// TIA Portal V18 export
FUNCTION_BLOCK "NG"   // FB2901, LAD
{ S7_Optimized_Access := 'TRUE' }
// stored: AutoNumber false, MemoryReserve 100, SetENOAutomatically false
   VAR
      NG_L_1 : "NGStatus";
      NG_L_2 { S7_SetPoint := 'True'} : "NGStatus";
      NG_L_3 { S7_SetPoint := 'True'} : "NGStatus";
      NG_UL_1 { S7_SetPoint := 'True'} : "NGStatus";
      NG_UL_2 { S7_SetPoint := 'True'} : "NGStatus";
      NG_UL_3 { S7_SetPoint := 'True'} : "NGStatus";
   END_VAR
   VAR_TEMP   // added for the SCL form of the ladder/FBD networks
      _w1 : Bool;
      _w2 : Bool;
      _w3 : Bool;
      _w4 : Bool;
      _w5 : Bool;
      _w6 : Bool;
      _w7 : Bool;
      _w8 : Bool;
      _w9 : Bool;
      _w10 : Bool;
      _w11 : Bool;
      _w12 : Bool;
      _w13 : Bool;
   END_VAR
BEGIN

REGION Network 1 (SCL): Input
   // NG1
   "PalletNGData".LoadingNGPallet.NG_1_1 := "iE1-UnloadingShaftPressNG_5";
   "PalletNGData".LoadingNGPallet.NG_1_2 := "iE1-UnloadingShaftPressNG_4";
   "PalletNGData".LoadingNGPallet.NG_1_3 := "iE1-UnloadingShaftPressNG_3";
   "PalletNGData".LoadingNGPallet.NG_1_4 := "iE1-UnloadingShaftPressNG_2";
   "PalletNGData".LoadingNGPallet.NG_1_5 := "iE1-UnloadingShaftPressNG_1";

   "PalletNGData".LoadingNGPallet.NG_2_1 := "iE1-UnloadingShaftScanNG_5";
   "PalletNGData".LoadingNGPallet.NG_2_2 := "iE1-UnloadingShaftScanNG_4";
   "PalletNGData".LoadingNGPallet.NG_2_3 := "iE1-UnloadingShaftScanNG_3";
   "PalletNGData".LoadingNGPallet.NG_2_4 := "iE1-UnloadingShaftScanNG_2";
   "PalletNGData".LoadingNGPallet.NG_2_5 := "iE1-UnloadingShaftScanNG_1";

   "PalletNGData".LoadingNGPallet.NG_3_1 := "iE1-UnloadingRingScanNG_5";
   "PalletNGData".LoadingNGPallet.NG_3_2 := "iE1-UnloadingRingScanNG_4";
   "PalletNGData".LoadingNGPallet.NG_3_3 := "iE1-UnloadingRingScanNG_3";
   "PalletNGData".LoadingNGPallet.NG_3_4 := "iE1-UnloadingRingScanNG_2";
   "PalletNGData".LoadingNGPallet.NG_3_5 := "iE1-UnloadingRingScanNG_1";

   // NG2
   "PalletNGData".UnLoadingNGPallet.NG_1_1 := "iE2-UnloadingPressNG_5";
   "PalletNGData".UnLoadingNGPallet.NG_1_2 := "iE2-UnloadingPressNG_4";
   "PalletNGData".UnLoadingNGPallet.NG_1_3 := "iE2-UnloadingPressNG_3";
   "PalletNGData".UnLoadingNGPallet.NG_1_4 := "iE2-UnloadingPressNG_2";
   "PalletNGData".UnLoadingNGPallet.NG_1_5 := "iE2-UnloadingPressNG_1";

   "PalletNGData".UnLoadingNGPallet.NG_2_1 := "iE2-UnloadingMagentScanNG_5";
   "PalletNGData".UnLoadingNGPallet.NG_2_2 := "iE2-UnloadingMagentScanNG_4";
   "PalletNGData".UnLoadingNGPallet.NG_2_3 := "iE2-UnloadingMagentScanNG_3";
   "PalletNGData".UnLoadingNGPallet.NG_2_4 := "iE2-UnloadingMagentScanNG_2";
   "PalletNGData".UnLoadingNGPallet.NG_2_5 := "iE2-UnloadingMagentScanNG_1";

   "PalletNGData".UnLoadingNGPallet.NG_3_1 := "iE2-UnloadingRingScanNG_5";
   "PalletNGData".UnLoadingNGPallet.NG_3_2 := "iE2-UnloadingRingScanNG_4";
   "PalletNGData".UnLoadingNGPallet.NG_3_3 := "iE2-UnloadingRingScanNG_3";
   "PalletNGData".UnLoadingNGPallet.NG_3_4 := "iE2-UnloadingRingScanNG_2";
   "PalletNGData".UnLoadingNGPallet.NG_3_5 := "iE2-UnloadingRingScanNG_1";
END_REGION

REGION Network 2: --------------------------------------- Load -------------------------------------------------------
END_REGION

REGION Network 3: Press
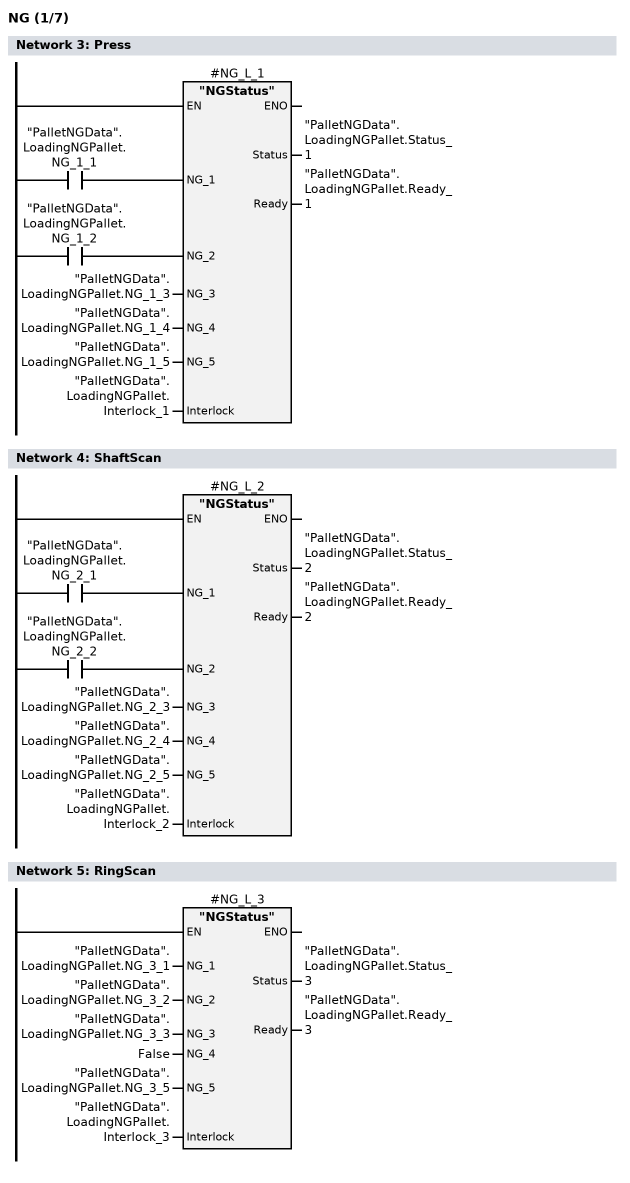
   RUNG wire#powerrail
      #NG_L_1(NG_1 := wire#w1, NG_2 := wire#w2, NG_3 := "PalletNGData".LoadingNGPallet.NG_1_3, NG_4 := "PalletNGData".LoadingNGPallet.NG_1_4, NG_5 := "PalletNGData".LoadingNGPallet.NG_1_5, Interlock := "PalletNGData".LoadingNGPallet.Interlock_1, Status => "PalletNGData".LoadingNGPallet.Status_1, Ready => "PalletNGData".LoadingNGPallet.Ready_1)
   END_RUNG
   RUNG wire#powerrail
      Contact( "PalletNGData".LoadingNGPallet.NG_1_1 )
   END_RUNG wire#w1
   RUNG wire#powerrail
      Contact( "PalletNGData".LoadingNGPallet.NG_1_2 )
   END_RUNG wire#w2
   // the same network as SCL:
   #NG_L_1(NG_1 := "PalletNGData".LoadingNGPallet.NG_1_1,   // "NGStatus"
           NG_2 := "PalletNGData".LoadingNGPallet.NG_1_2,
           NG_3 := "PalletNGData".LoadingNGPallet.NG_1_3,
           NG_4 := "PalletNGData".LoadingNGPallet.NG_1_4,
           NG_5 := "PalletNGData".LoadingNGPallet.NG_1_5,
           Interlock := "PalletNGData".LoadingNGPallet.Interlock_1,
           Status => "PalletNGData".LoadingNGPallet.Status_1,
           Ready => "PalletNGData".LoadingNGPallet.Ready_1);
END_REGION

REGION Network 4: ShaftScan
   RUNG wire#powerrail
      #NG_L_2(NG_1 := wire#w1, NG_2 := wire#w2, NG_3 := "PalletNGData".LoadingNGPallet.NG_2_3, NG_4 := "PalletNGData".LoadingNGPallet.NG_2_4, NG_5 := "PalletNGData".LoadingNGPallet.NG_2_5, Interlock := "PalletNGData".LoadingNGPallet.Interlock_2, Status => "PalletNGData".LoadingNGPallet.Status_2, Ready => "PalletNGData".LoadingNGPallet.Ready_2)
   END_RUNG
   RUNG wire#powerrail
      Contact( "PalletNGData".LoadingNGPallet.NG_2_1 )
   END_RUNG wire#w1
   RUNG wire#powerrail
      Contact( "PalletNGData".LoadingNGPallet.NG_2_2 )
   END_RUNG wire#w2
   // the same network as SCL:
   #NG_L_2(NG_1 := "PalletNGData".LoadingNGPallet.NG_2_1,   // "NGStatus"
           NG_2 := "PalletNGData".LoadingNGPallet.NG_2_2,
           NG_3 := "PalletNGData".LoadingNGPallet.NG_2_3,
           NG_4 := "PalletNGData".LoadingNGPallet.NG_2_4,
           NG_5 := "PalletNGData".LoadingNGPallet.NG_2_5,
           Interlock := "PalletNGData".LoadingNGPallet.Interlock_2,
           Status => "PalletNGData".LoadingNGPallet.Status_2,
           Ready => "PalletNGData".LoadingNGPallet.Ready_2);
END_REGION

REGION Network 5: RingScan
   RUNG wire#powerrail
      #NG_L_3(NG_1 := "PalletNGData".LoadingNGPallet.NG_3_1, NG_2 := "PalletNGData".LoadingNGPallet.NG_3_2, NG_3 := "PalletNGData".LoadingNGPallet.NG_3_3, NG_4 := False, NG_5 := "PalletNGData".LoadingNGPallet.NG_3_5, Interlock := "PalletNGData".LoadingNGPallet.Interlock_3, Status => "PalletNGData".LoadingNGPallet.Status_3, Ready => "PalletNGData".LoadingNGPallet.Ready_3)
   END_RUNG
   // the same network as SCL:
   #NG_L_3(NG_1 := "PalletNGData".LoadingNGPallet.NG_3_1,   // "NGStatus"
           NG_2 := "PalletNGData".LoadingNGPallet.NG_3_2,
           NG_3 := "PalletNGData".LoadingNGPallet.NG_3_3,
           NG_4 := False,
           NG_5 := "PalletNGData".LoadingNGPallet.NG_3_5,
           Interlock := "PalletNGData".LoadingNGPallet.Interlock_3,
           Status => "PalletNGData".LoadingNGPallet.Status_3,
           Ready => "PalletNGData".LoadingNGPallet.Ready_3);
END_REGION

REGION Network 6: InterLock
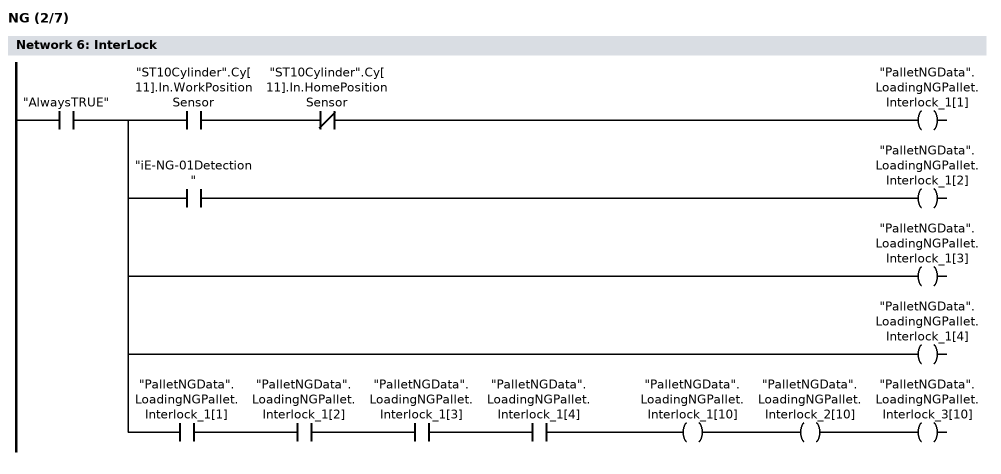
   RUNG wire#powerrail
      Contact( "AlwaysTRUE" )
      wire#w1
      Contact( "ST10Cylinder".Cy[11].In.WorkPositionSensor )
      I_Contact( "ST10Cylinder".Cy[11].In.HomePositionSensor )
      Coil( "PalletNGData".LoadingNGPallet.Interlock_1[1] )
   END_RUNG
   RUNG wire#w1
      Contact( "iE-NG-01Detection" )
      Coil( "PalletNGData".LoadingNGPallet.Interlock_1[2] )
   END_RUNG
   RUNG wire#w1
      Coil( "PalletNGData".LoadingNGPallet.Interlock_1[3] )
   END_RUNG
   RUNG wire#w1
      Coil( "PalletNGData".LoadingNGPallet.Interlock_1[4] )
   END_RUNG
   RUNG wire#w1
      Contact( "PalletNGData".LoadingNGPallet.Interlock_1[1] )
      Contact( "PalletNGData".LoadingNGPallet.Interlock_1[2] )
      Contact( "PalletNGData".LoadingNGPallet.Interlock_1[3] )
      Contact( "PalletNGData".LoadingNGPallet.Interlock_1[4] )
      Coil( "PalletNGData".LoadingNGPallet.Interlock_1[10] )
      Coil( "PalletNGData".LoadingNGPallet.Interlock_2[10] )
      Coil( "PalletNGData".LoadingNGPallet.Interlock_3[10] )
   END_RUNG
   // the same network as SCL:
   "PalletNGData".LoadingNGPallet.Interlock_1[1] := "AlwaysTRUE" AND "ST10Cylinder".Cy[11].In.WorkPositionSensor AND NOT "ST10Cylinder".Cy[11].In.HomePositionSensor;
   "PalletNGData".LoadingNGPallet.Interlock_1[2] := "AlwaysTRUE" AND "iE-NG-01Detection";
   "PalletNGData".LoadingNGPallet.Interlock_1[3] := "AlwaysTRUE";
   "PalletNGData".LoadingNGPallet.Interlock_1[4] := "AlwaysTRUE";
   #_w1 := "AlwaysTRUE" AND "PalletNGData".LoadingNGPallet.Interlock_1[1] AND "PalletNGData".LoadingNGPallet.Interlock_1[2] AND "PalletNGData".LoadingNGPallet.Interlock_1[3] AND "PalletNGData".LoadingNGPallet.Interlock_1[4];
   "PalletNGData".LoadingNGPallet.Interlock_1[10] := #_w1;
   "PalletNGData".LoadingNGPallet.Interlock_2[10] := #_w1;
   "PalletNGData".LoadingNGPallet.Interlock_3[10] := #_w1;
END_REGION

REGION Network 7: NG_Button
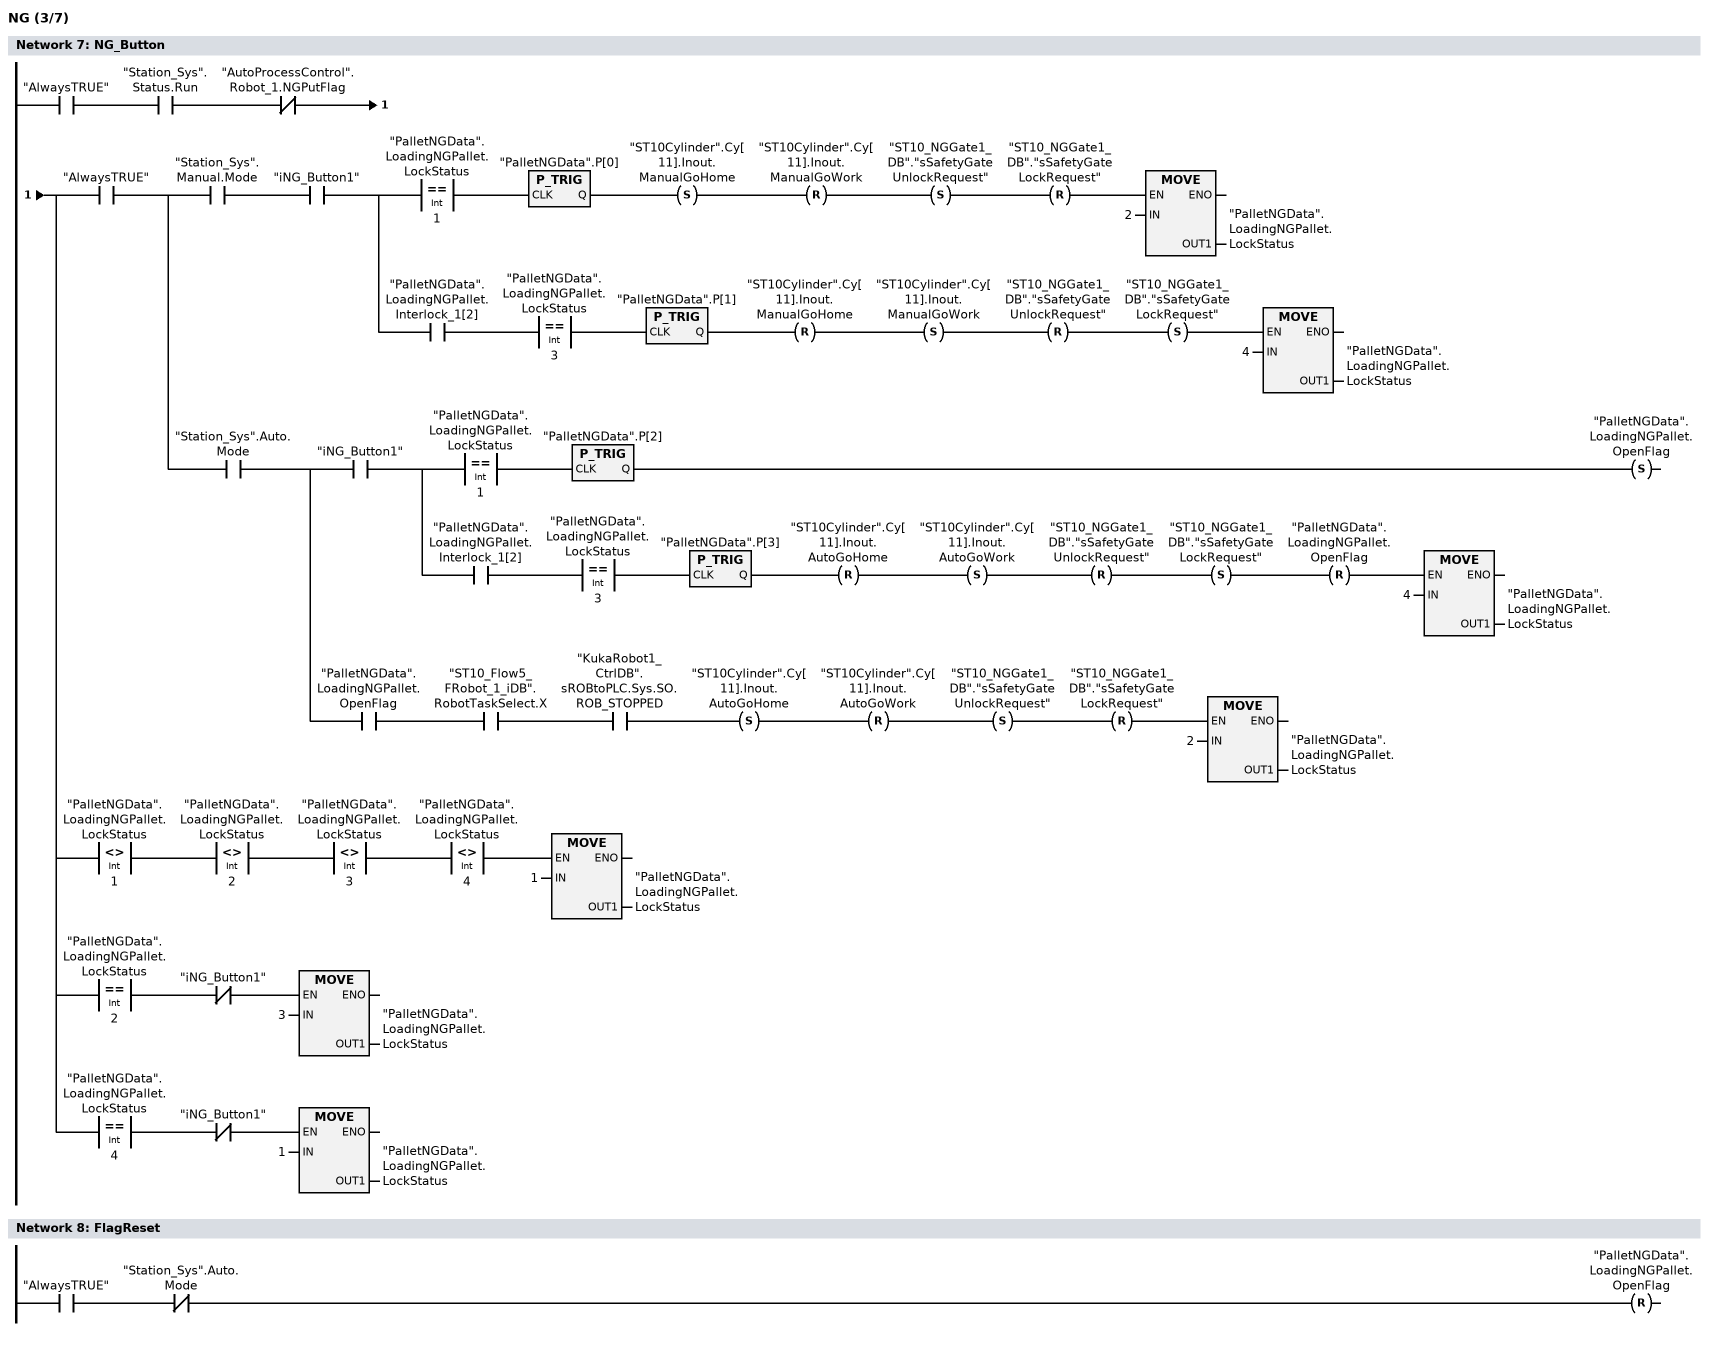
   RUNG wire#powerrail
      Contact( "AlwaysTRUE" )
      Contact( "Station_Sys".Status.Run )
      I_Contact( "AutoProcessControl".Robot_1.NGPutFlag )
      wire#w1
      Contact( "AlwaysTRUE" )
      wire#w2
      Contact( "Station_Sys".Manual.Mode )
      Contact( "iNG_Button1" )
      wire#w3
      { S7_Templates := "SrcType := Int" } EQ_Contact(in1 := "PalletNGData".LoadingNGPallet.LockStatus, in2 := 1)
      P_Trig( "PalletNGData".P[0] )
      S_Coil( "ST10Cylinder".Cy[11].Inout.ManualGoHome )
      R_Coil( "ST10Cylinder".Cy[11].Inout.ManualGoWork )
      S_Coil( "ST10_NGGate1_DB"."sSafetyGate UnlockRequest" )
      R_Coil( "ST10_NGGate1_DB"."sSafetyGate LockRequest" )
      Move(in := 2, out1 => "PalletNGData".LoadingNGPallet.LockStatus)
   END_RUNG
   RUNG wire#w3
      Contact( "PalletNGData".LoadingNGPallet.Interlock_1[2] )
      { S7_Templates := "SrcType := Int" } EQ_Contact(in1 := "PalletNGData".LoadingNGPallet.LockStatus, in2 := 3)
      P_Trig( "PalletNGData".P[1] )
      R_Coil( "ST10Cylinder".Cy[11].Inout.ManualGoHome )
      S_Coil( "ST10Cylinder".Cy[11].Inout.ManualGoWork )
      R_Coil( "ST10_NGGate1_DB"."sSafetyGate UnlockRequest" )
      S_Coil( "ST10_NGGate1_DB"."sSafetyGate LockRequest" )
      Move(in := 4, out1 => "PalletNGData".LoadingNGPallet.LockStatus)
   END_RUNG
   RUNG wire#w2
      Contact( "Station_Sys".Auto.Mode )
      wire#w4
      Contact( "iNG_Button1" )
      wire#w5
      { S7_Templates := "SrcType := Int" } EQ_Contact(in1 := "PalletNGData".LoadingNGPallet.LockStatus, in2 := 1)
      P_Trig( "PalletNGData".P[2] )
      S_Coil( "PalletNGData".LoadingNGPallet.OpenFlag )
   END_RUNG
   RUNG wire#w5
      Contact( "PalletNGData".LoadingNGPallet.Interlock_1[2] )
      { S7_Templates := "SrcType := Int" } EQ_Contact(in1 := "PalletNGData".LoadingNGPallet.LockStatus, in2 := 3)
      P_Trig( "PalletNGData".P[3] )
      R_Coil( "ST10Cylinder".Cy[11].Inout.AutoGoHome )
      S_Coil( "ST10Cylinder".Cy[11].Inout.AutoGoWork )
      R_Coil( "ST10_NGGate1_DB"."sSafetyGate UnlockRequest" )
      S_Coil( "ST10_NGGate1_DB"."sSafetyGate LockRequest" )
      R_Coil( "PalletNGData".LoadingNGPallet.OpenFlag )
      Move(in := 4, out1 => "PalletNGData".LoadingNGPallet.LockStatus)
   END_RUNG
   RUNG wire#w4
      Contact( "PalletNGData".LoadingNGPallet.OpenFlag )
      Contact( "ST10_Flow5_FRobot_1_iDB".RobotTaskSelect.X )
      Contact( "KukaRobot1_CtrlDB".sROBtoPLC.Sys.SO.ROB_STOPPED )
      S_Coil( "ST10Cylinder".Cy[11].Inout.AutoGoHome )
      R_Coil( "ST10Cylinder".Cy[11].Inout.AutoGoWork )
      S_Coil( "ST10_NGGate1_DB"."sSafetyGate UnlockRequest" )
      R_Coil( "ST10_NGGate1_DB"."sSafetyGate LockRequest" )
      Move(in := 2, out1 => "PalletNGData".LoadingNGPallet.LockStatus)
   END_RUNG
   RUNG wire#w1
      { S7_Templates := "SrcType := Int" } NE_Contact(in1 := "PalletNGData".LoadingNGPallet.LockStatus, in2 := 1)
      { S7_Templates := "SrcType := Int" } NE_Contact(in1 := "PalletNGData".LoadingNGPallet.LockStatus, in2 := 2)
      { S7_Templates := "SrcType := Int" } NE_Contact(in1 := "PalletNGData".LoadingNGPallet.LockStatus, in2 := 3)
      { S7_Templates := "SrcType := Int" } NE_Contact(in1 := "PalletNGData".LoadingNGPallet.LockStatus, in2 := 4)
      Move(in := 1, out1 => "PalletNGData".LoadingNGPallet.LockStatus)
   END_RUNG
   RUNG wire#w1
      { S7_Templates := "SrcType := Int" } EQ_Contact(in1 := "PalletNGData".LoadingNGPallet.LockStatus, in2 := 2)
      I_Contact( "iNG_Button1" )
      Move(in := 3, out1 => "PalletNGData".LoadingNGPallet.LockStatus)
   END_RUNG
   RUNG wire#w1
      { S7_Templates := "SrcType := Int" } EQ_Contact(in1 := "PalletNGData".LoadingNGPallet.LockStatus, in2 := 4)
      I_Contact( "iNG_Button1" )
      Move(in := 1, out1 => "PalletNGData".LoadingNGPallet.LockStatus)
   END_RUNG
   // the same network as SCL:
   #_w1 := "AlwaysTRUE" AND "Station_Sys".Status.Run AND NOT "AutoProcessControl".Robot_1.NGPutFlag;
   #_w2 := #_w1 AND "AlwaysTRUE";
   #_w3 := #_w2 AND "Station_Sys".Manual.Mode AND "iNG_Button1";
   #_w4 := #_w3 AND ("PalletNGData".LoadingNGPallet.LockStatus = 1);
   #_w5 := #_w4 AND NOT "PalletNGData".P[0];   // rising edge
   "PalletNGData".P[0] := #_w4;
   IF #_w5 THEN
       "ST10Cylinder".Cy[11].Inout.ManualGoHome := TRUE;
       "ST10Cylinder".Cy[11].Inout.ManualGoWork := FALSE;
       "ST10_NGGate1_DB"."sSafetyGate UnlockRequest" := TRUE;
       "ST10_NGGate1_DB"."sSafetyGate LockRequest" := FALSE;
       "PalletNGData".LoadingNGPallet.LockStatus := 2;
   END_IF;
   #_w6 := #_w3 AND "PalletNGData".LoadingNGPallet.Interlock_1[2] AND ("PalletNGData".LoadingNGPallet.LockStatus = 3);
   #_w7 := #_w6 AND NOT "PalletNGData".P[1];   // rising edge
   "PalletNGData".P[1] := #_w6;
   IF #_w7 THEN
       "ST10Cylinder".Cy[11].Inout.ManualGoHome := FALSE;
       "ST10Cylinder".Cy[11].Inout.ManualGoWork := TRUE;
       "ST10_NGGate1_DB"."sSafetyGate UnlockRequest" := FALSE;
       "ST10_NGGate1_DB"."sSafetyGate LockRequest" := TRUE;
       "PalletNGData".LoadingNGPallet.LockStatus := 4;
   END_IF;
   #_w8 := #_w2 AND "Station_Sys".Auto.Mode;
   #_w9 := #_w8 AND "iNG_Button1";
   #_w10 := #_w9 AND ("PalletNGData".LoadingNGPallet.LockStatus = 1);
   #_w11 := #_w10 AND NOT "PalletNGData".P[2];   // rising edge
   "PalletNGData".P[2] := #_w10;
   IF #_w11 THEN "PalletNGData".LoadingNGPallet.OpenFlag := TRUE; END_IF;
   #_w12 := #_w9 AND "PalletNGData".LoadingNGPallet.Interlock_1[2] AND ("PalletNGData".LoadingNGPallet.LockStatus = 3);
   #_w13 := #_w12 AND NOT "PalletNGData".P[3];   // rising edge
   "PalletNGData".P[3] := #_w12;
   IF #_w13 THEN
       "ST10Cylinder".Cy[11].Inout.AutoGoHome := FALSE;
       "ST10Cylinder".Cy[11].Inout.AutoGoWork := TRUE;
       "ST10_NGGate1_DB"."sSafetyGate UnlockRequest" := FALSE;
       "ST10_NGGate1_DB"."sSafetyGate LockRequest" := TRUE;
       "PalletNGData".LoadingNGPallet.OpenFlag := FALSE;
       "PalletNGData".LoadingNGPallet.LockStatus := 4;
   END_IF;
   IF #_w8 AND "PalletNGData".LoadingNGPallet.OpenFlag AND "ST10_Flow5_FRobot_1_iDB".RobotTaskSelect.X AND "KukaRobot1_CtrlDB".sROBtoPLC.Sys.SO.ROB_STOPPED THEN
       "ST10Cylinder".Cy[11].Inout.AutoGoHome := TRUE;
       "ST10Cylinder".Cy[11].Inout.AutoGoWork := FALSE;
       "ST10_NGGate1_DB"."sSafetyGate UnlockRequest" := TRUE;
       "ST10_NGGate1_DB"."sSafetyGate LockRequest" := FALSE;
       "PalletNGData".LoadingNGPallet.LockStatus := 2;
   END_IF;
   IF #_w1 AND ("PalletNGData".LoadingNGPallet.LockStatus <> 1) AND ("PalletNGData".LoadingNGPallet.LockStatus <> 2) AND ("PalletNGData".LoadingNGPallet.LockStatus <> 3) AND ("PalletNGData".LoadingNGPallet.LockStatus <> 4) THEN
       "PalletNGData".LoadingNGPallet.LockStatus := 1;
   END_IF;
   IF #_w1 AND ("PalletNGData".LoadingNGPallet.LockStatus = 2) AND NOT "iNG_Button1" THEN
       "PalletNGData".LoadingNGPallet.LockStatus := 3;
   END_IF;
   IF #_w1 AND ("PalletNGData".LoadingNGPallet.LockStatus = 4) AND NOT "iNG_Button1" THEN
       "PalletNGData".LoadingNGPallet.LockStatus := 1;
   END_IF;
END_REGION

REGION Network 8: FlagReset
   RUNG wire#powerrail
      Contact( "AlwaysTRUE" )
      I_Contact( "Station_Sys".Auto.Mode )
      R_Coil( "PalletNGData".LoadingNGPallet.OpenFlag )
   END_RUNG
   // the same network as SCL:
   IF "AlwaysTRUE" AND NOT "Station_Sys".Auto.Mode THEN
       "PalletNGData".LoadingNGPallet.OpenFlag := FALSE;
   END_IF;
END_REGION

REGION Network 9: NG Door
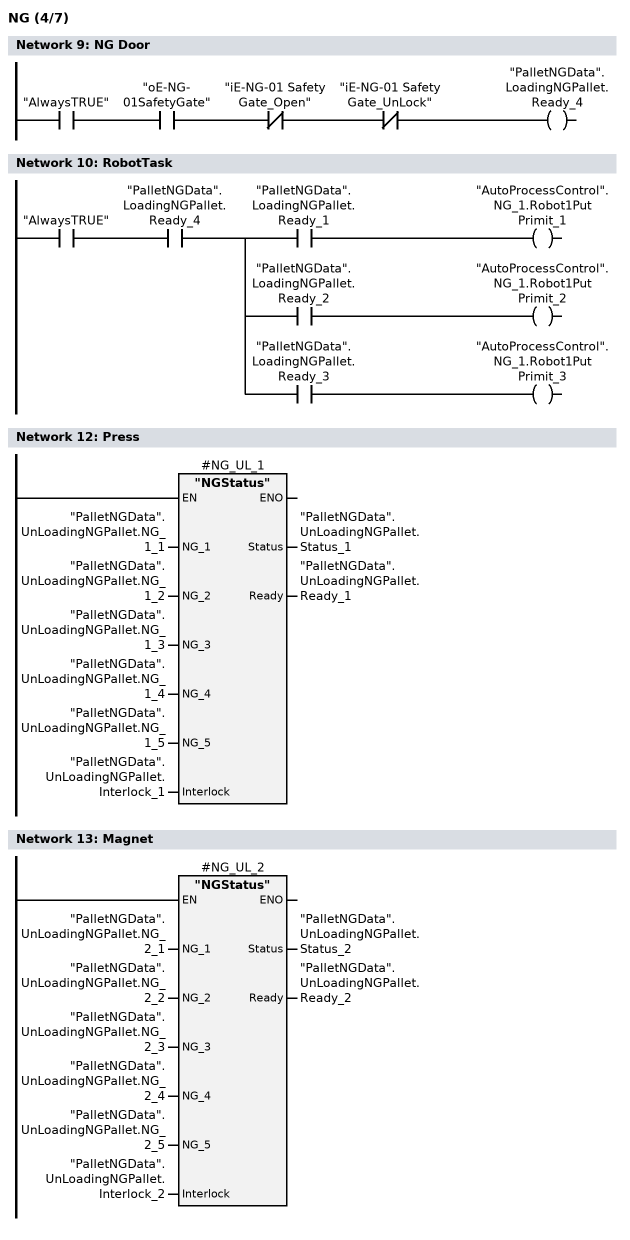
   RUNG wire#powerrail
      Contact( "AlwaysTRUE" )
      Contact( "oE-NG-01SafetyGate" )
      I_Contact( "iE-NG-01 Safety Gate_Open" )
      I_Contact( "iE-NG-01 Safety Gate_UnLock" )
      Coil( "PalletNGData".LoadingNGPallet.Ready_4 )
   END_RUNG
   // the same network as SCL:
   "PalletNGData".LoadingNGPallet.Ready_4 := "AlwaysTRUE" AND "oE-NG-01SafetyGate" AND NOT "iE-NG-01 Safety Gate_Open" AND NOT "iE-NG-01 Safety Gate_UnLock";
END_REGION

REGION Network 10: RobotTask
   RUNG wire#powerrail
      Contact( "AlwaysTRUE" )
      Contact( "PalletNGData".LoadingNGPallet.Ready_4 )
      wire#w1
      Contact( "PalletNGData".LoadingNGPallet.Ready_1 )
      Coil( "AutoProcessControl".NG_1.Robot1PutPrimit_1 )
   END_RUNG
   RUNG wire#w1
      Contact( "PalletNGData".LoadingNGPallet.Ready_2 )
      Coil( "AutoProcessControl".NG_1.Robot1PutPrimit_2 )
   END_RUNG
   RUNG wire#w1
      Contact( "PalletNGData".LoadingNGPallet.Ready_3 )
      Coil( "AutoProcessControl".NG_1.Robot1PutPrimit_3 )
   END_RUNG
   // the same network as SCL:
   #_w1 := "AlwaysTRUE" AND "PalletNGData".LoadingNGPallet.Ready_4;
   "AutoProcessControl".NG_1.Robot1PutPrimit_1 := #_w1 AND "PalletNGData".LoadingNGPallet.Ready_1;
   "AutoProcessControl".NG_1.Robot1PutPrimit_2 := #_w1 AND "PalletNGData".LoadingNGPallet.Ready_2;
   "AutoProcessControl".NG_1.Robot1PutPrimit_3 := #_w1 AND "PalletNGData".LoadingNGPallet.Ready_3;
END_REGION

REGION Network 11: --------------------------------------- UnLoad -------------------------------------------------------
END_REGION

REGION Network 12: Press
   RUNG wire#powerrail
      #NG_UL_1(NG_1 := "PalletNGData".UnLoadingNGPallet.NG_1_1, NG_2 := "PalletNGData".UnLoadingNGPallet.NG_1_2, NG_3 := "PalletNGData".UnLoadingNGPallet.NG_1_3, NG_4 := "PalletNGData".UnLoadingNGPallet.NG_1_4, NG_5 := "PalletNGData".UnLoadingNGPallet.NG_1_5, Interlock := "PalletNGData".UnLoadingNGPallet.Interlock_1, Status => "PalletNGData".UnLoadingNGPallet.Status_1, Ready => "PalletNGData".UnLoadingNGPallet.Ready_1)
   END_RUNG
   // the same network as SCL:
   #NG_UL_1(NG_1 := "PalletNGData".UnLoadingNGPallet.NG_1_1,   // "NGStatus"
            NG_2 := "PalletNGData".UnLoadingNGPallet.NG_1_2,
            NG_3 := "PalletNGData".UnLoadingNGPallet.NG_1_3,
            NG_4 := "PalletNGData".UnLoadingNGPallet.NG_1_4,
            NG_5 := "PalletNGData".UnLoadingNGPallet.NG_1_5,
            Interlock := "PalletNGData".UnLoadingNGPallet.Interlock_1,
            Status => "PalletNGData".UnLoadingNGPallet.Status_1,
            Ready => "PalletNGData".UnLoadingNGPallet.Ready_1);
END_REGION

REGION Network 13: Magnet
   RUNG wire#powerrail
      #NG_UL_2(NG_1 := "PalletNGData".UnLoadingNGPallet.NG_2_1, NG_2 := "PalletNGData".UnLoadingNGPallet.NG_2_2, NG_3 := "PalletNGData".UnLoadingNGPallet.NG_2_3, NG_4 := "PalletNGData".UnLoadingNGPallet.NG_2_4, NG_5 := "PalletNGData".UnLoadingNGPallet.NG_2_5, Interlock := "PalletNGData".UnLoadingNGPallet.Interlock_2, Status => "PalletNGData".UnLoadingNGPallet.Status_2, Ready => "PalletNGData".UnLoadingNGPallet.Ready_2)
   END_RUNG
   // the same network as SCL:
   #NG_UL_2(NG_1 := "PalletNGData".UnLoadingNGPallet.NG_2_1,   // "NGStatus"
            NG_2 := "PalletNGData".UnLoadingNGPallet.NG_2_2,
            NG_3 := "PalletNGData".UnLoadingNGPallet.NG_2_3,
            NG_4 := "PalletNGData".UnLoadingNGPallet.NG_2_4,
            NG_5 := "PalletNGData".UnLoadingNGPallet.NG_2_5,
            Interlock := "PalletNGData".UnLoadingNGPallet.Interlock_2,
            Status => "PalletNGData".UnLoadingNGPallet.Status_2,
            Ready => "PalletNGData".UnLoadingNGPallet.Ready_2);
END_REGION

REGION Network 14: Ring
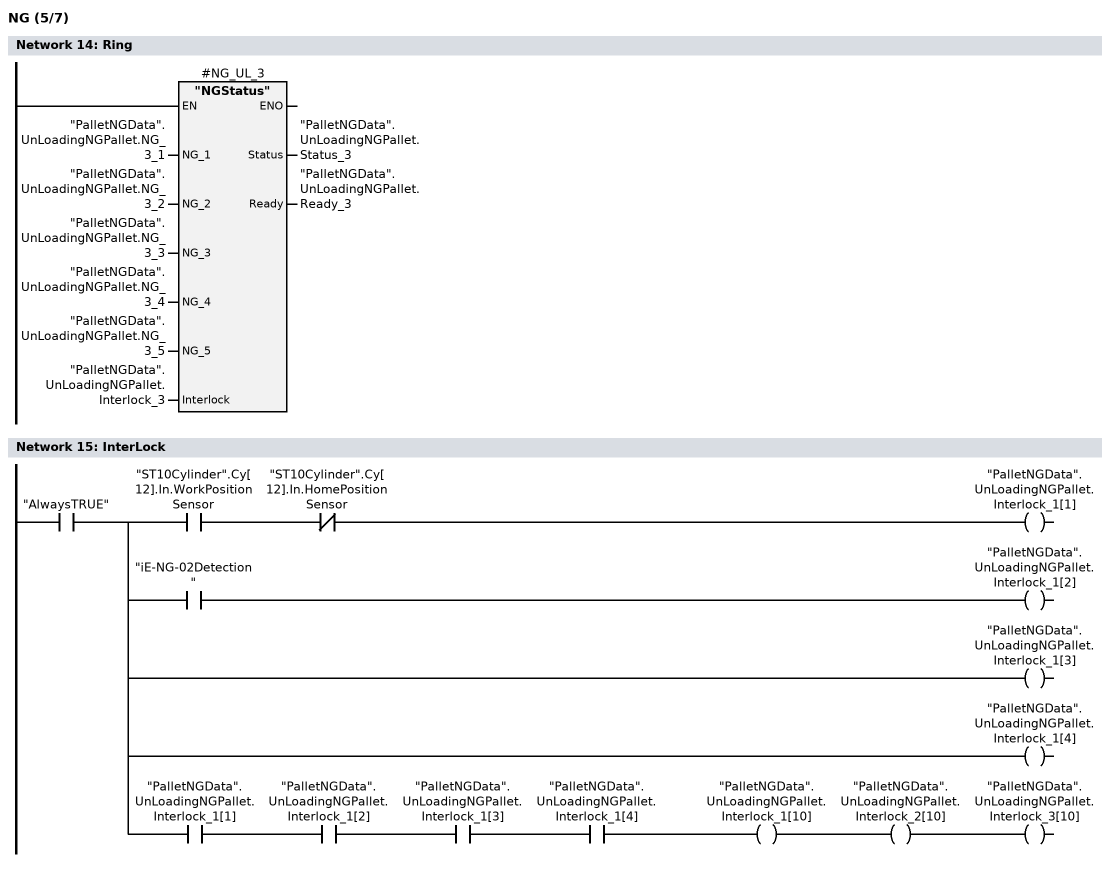
   RUNG wire#powerrail
      #NG_UL_3(NG_1 := "PalletNGData".UnLoadingNGPallet.NG_3_1, NG_2 := "PalletNGData".UnLoadingNGPallet.NG_3_2, NG_3 := "PalletNGData".UnLoadingNGPallet.NG_3_3, NG_4 := "PalletNGData".UnLoadingNGPallet.NG_3_4, NG_5 := "PalletNGData".UnLoadingNGPallet.NG_3_5, Interlock := "PalletNGData".UnLoadingNGPallet.Interlock_3, Status => "PalletNGData".UnLoadingNGPallet.Status_3, Ready => "PalletNGData".UnLoadingNGPallet.Ready_3)
   END_RUNG
   // the same network as SCL:
   #NG_UL_3(NG_1 := "PalletNGData".UnLoadingNGPallet.NG_3_1,   // "NGStatus"
            NG_2 := "PalletNGData".UnLoadingNGPallet.NG_3_2,
            NG_3 := "PalletNGData".UnLoadingNGPallet.NG_3_3,
            NG_4 := "PalletNGData".UnLoadingNGPallet.NG_3_4,
            NG_5 := "PalletNGData".UnLoadingNGPallet.NG_3_5,
            Interlock := "PalletNGData".UnLoadingNGPallet.Interlock_3,
            Status => "PalletNGData".UnLoadingNGPallet.Status_3,
            Ready => "PalletNGData".UnLoadingNGPallet.Ready_3);
END_REGION

REGION Network 15: InterLock
   RUNG wire#powerrail
      Contact( "AlwaysTRUE" )
      wire#w1
      Contact( "ST10Cylinder".Cy[12].In.WorkPositionSensor )
      I_Contact( "ST10Cylinder".Cy[12].In.HomePositionSensor )
      Coil( "PalletNGData".UnLoadingNGPallet.Interlock_1[1] )
   END_RUNG
   RUNG wire#w1
      Contact( "iE-NG-02Detection" )
      Coil( "PalletNGData".UnLoadingNGPallet.Interlock_1[2] )
   END_RUNG
   RUNG wire#w1
      Coil( "PalletNGData".UnLoadingNGPallet.Interlock_1[3] )
   END_RUNG
   RUNG wire#w1
      Coil( "PalletNGData".UnLoadingNGPallet.Interlock_1[4] )
   END_RUNG
   RUNG wire#w1
      Contact( "PalletNGData".UnLoadingNGPallet.Interlock_1[1] )
      Contact( "PalletNGData".UnLoadingNGPallet.Interlock_1[2] )
      Contact( "PalletNGData".UnLoadingNGPallet.Interlock_1[3] )
      Contact( "PalletNGData".UnLoadingNGPallet.Interlock_1[4] )
      Coil( "PalletNGData".UnLoadingNGPallet.Interlock_1[10] )
      Coil( "PalletNGData".UnLoadingNGPallet.Interlock_2[10] )
      Coil( "PalletNGData".UnLoadingNGPallet.Interlock_3[10] )
   END_RUNG
   // the same network as SCL:
   "PalletNGData".UnLoadingNGPallet.Interlock_1[1] := "AlwaysTRUE" AND "ST10Cylinder".Cy[12].In.WorkPositionSensor AND NOT "ST10Cylinder".Cy[12].In.HomePositionSensor;
   "PalletNGData".UnLoadingNGPallet.Interlock_1[2] := "AlwaysTRUE" AND "iE-NG-02Detection";
   "PalletNGData".UnLoadingNGPallet.Interlock_1[3] := "AlwaysTRUE";
   "PalletNGData".UnLoadingNGPallet.Interlock_1[4] := "AlwaysTRUE";
   #_w1 := "AlwaysTRUE" AND "PalletNGData".UnLoadingNGPallet.Interlock_1[1] AND "PalletNGData".UnLoadingNGPallet.Interlock_1[2] AND "PalletNGData".UnLoadingNGPallet.Interlock_1[3] AND "PalletNGData".UnLoadingNGPallet.Interlock_1[4];
   "PalletNGData".UnLoadingNGPallet.Interlock_1[10] := #_w1;
   "PalletNGData".UnLoadingNGPallet.Interlock_2[10] := #_w1;
   "PalletNGData".UnLoadingNGPallet.Interlock_3[10] := #_w1;
END_REGION

REGION Network 16: NG_Button
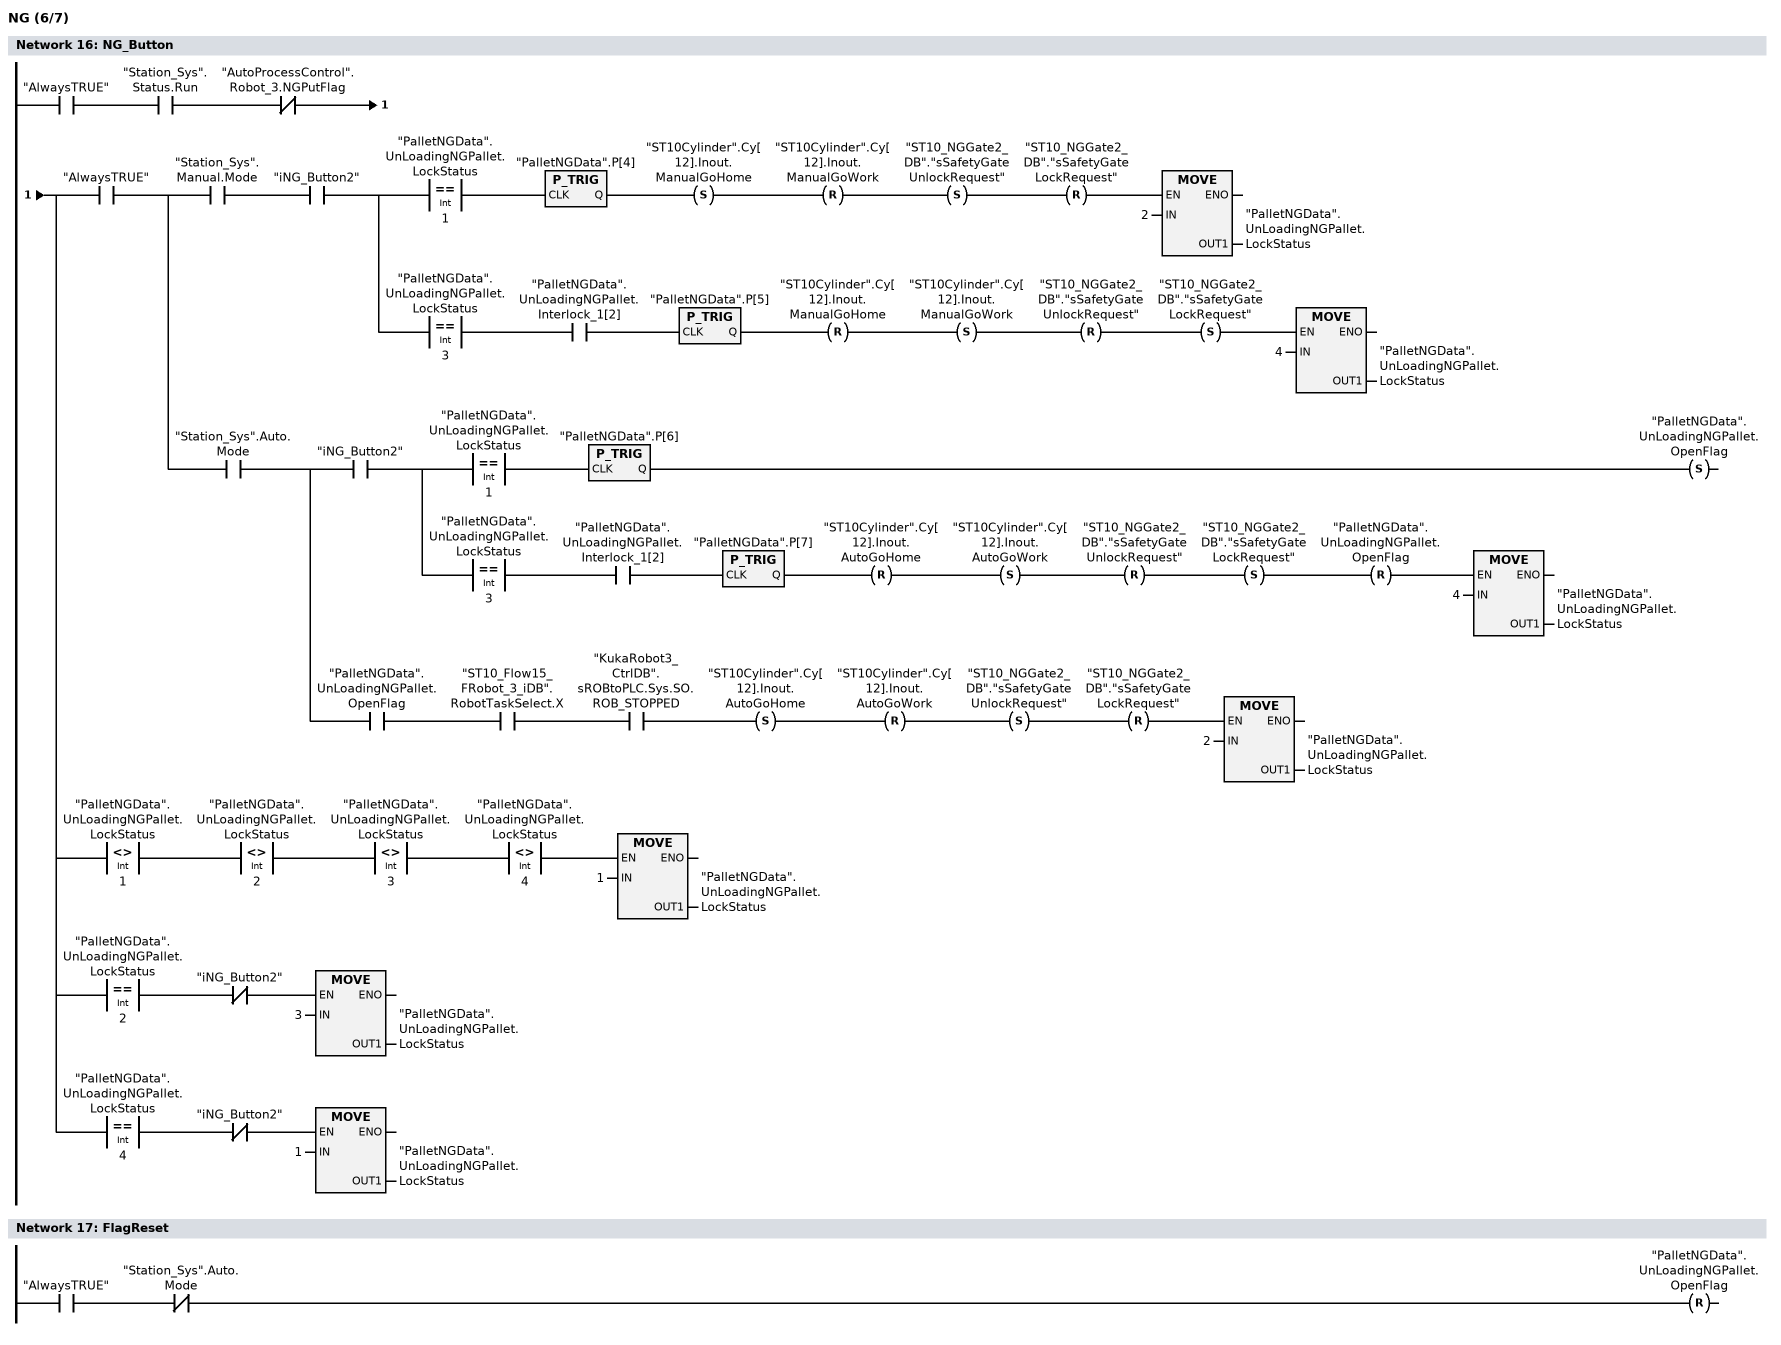
   RUNG wire#powerrail
      Contact( "AlwaysTRUE" )
      Contact( "Station_Sys".Status.Run )
      I_Contact( "AutoProcessControl".Robot_3.NGPutFlag )
      wire#w1
      Contact( "AlwaysTRUE" )
      wire#w2
      Contact( "Station_Sys".Manual.Mode )
      Contact( "iNG_Button2" )
      wire#w3
      { S7_Templates := "SrcType := Int" } EQ_Contact(in1 := "PalletNGData".UnLoadingNGPallet.LockStatus, in2 := 1)
      P_Trig( "PalletNGData".P[4] )
      S_Coil( "ST10Cylinder".Cy[12].Inout.ManualGoHome )
      R_Coil( "ST10Cylinder".Cy[12].Inout.ManualGoWork )
      S_Coil( "ST10_NGGate2_DB"."sSafetyGate UnlockRequest" )
      R_Coil( "ST10_NGGate2_DB"."sSafetyGate LockRequest" )
      Move(in := 2, out1 => "PalletNGData".UnLoadingNGPallet.LockStatus)
   END_RUNG
   RUNG wire#w3
      { S7_Templates := "SrcType := Int" } EQ_Contact(in1 := "PalletNGData".UnLoadingNGPallet.LockStatus, in2 := 3)
      Contact( "PalletNGData".UnLoadingNGPallet.Interlock_1[2] )
      P_Trig( "PalletNGData".P[5] )
      R_Coil( "ST10Cylinder".Cy[12].Inout.ManualGoHome )
      S_Coil( "ST10Cylinder".Cy[12].Inout.ManualGoWork )
      R_Coil( "ST10_NGGate2_DB"."sSafetyGate UnlockRequest" )
      S_Coil( "ST10_NGGate2_DB"."sSafetyGate LockRequest" )
      Move(in := 4, out1 => "PalletNGData".UnLoadingNGPallet.LockStatus)
   END_RUNG
   RUNG wire#w2
      Contact( "Station_Sys".Auto.Mode )
      wire#w4
      Contact( "iNG_Button2" )
      wire#w5
      { S7_Templates := "SrcType := Int" } EQ_Contact(in1 := "PalletNGData".UnLoadingNGPallet.LockStatus, in2 := 1)
      P_Trig( "PalletNGData".P[6] )
      S_Coil( "PalletNGData".UnLoadingNGPallet.OpenFlag )
   END_RUNG
   RUNG wire#w5
      { S7_Templates := "SrcType := Int" } EQ_Contact(in1 := "PalletNGData".UnLoadingNGPallet.LockStatus, in2 := 3)
      Contact( "PalletNGData".UnLoadingNGPallet.Interlock_1[2] )
      P_Trig( "PalletNGData".P[7] )
      R_Coil( "ST10Cylinder".Cy[12].Inout.AutoGoHome )
      S_Coil( "ST10Cylinder".Cy[12].Inout.AutoGoWork )
      R_Coil( "ST10_NGGate2_DB"."sSafetyGate UnlockRequest" )
      S_Coil( "ST10_NGGate2_DB"."sSafetyGate LockRequest" )
      R_Coil( "PalletNGData".UnLoadingNGPallet.OpenFlag )
      Move(in := 4, out1 => "PalletNGData".UnLoadingNGPallet.LockStatus)
   END_RUNG
   RUNG wire#w4
      Contact( "PalletNGData".UnLoadingNGPallet.OpenFlag )
      Contact( "ST10_Flow15_FRobot_3_iDB".RobotTaskSelect.X )
      Contact( "KukaRobot3_CtrlDB".sROBtoPLC.Sys.SO.ROB_STOPPED )
      S_Coil( "ST10Cylinder".Cy[12].Inout.AutoGoHome )
      R_Coil( "ST10Cylinder".Cy[12].Inout.AutoGoWork )
      S_Coil( "ST10_NGGate2_DB"."sSafetyGate UnlockRequest" )
      R_Coil( "ST10_NGGate2_DB"."sSafetyGate LockRequest" )
      Move(in := 2, out1 => "PalletNGData".UnLoadingNGPallet.LockStatus)
   END_RUNG
   RUNG wire#w1
      { S7_Templates := "SrcType := Int" } NE_Contact(in1 := "PalletNGData".UnLoadingNGPallet.LockStatus, in2 := 1)
      { S7_Templates := "SrcType := Int" } NE_Contact(in1 := "PalletNGData".UnLoadingNGPallet.LockStatus, in2 := 2)
      { S7_Templates := "SrcType := Int" } NE_Contact(in1 := "PalletNGData".UnLoadingNGPallet.LockStatus, in2 := 3)
      { S7_Templates := "SrcType := Int" } NE_Contact(in1 := "PalletNGData".UnLoadingNGPallet.LockStatus, in2 := 4)
      Move(in := 1, out1 => "PalletNGData".UnLoadingNGPallet.LockStatus)
   END_RUNG
   RUNG wire#w1
      { S7_Templates := "SrcType := Int" } EQ_Contact(in1 := "PalletNGData".UnLoadingNGPallet.LockStatus, in2 := 2)
      I_Contact( "iNG_Button2" )
      Move(in := 3, out1 => "PalletNGData".UnLoadingNGPallet.LockStatus)
   END_RUNG
   RUNG wire#w1
      { S7_Templates := "SrcType := Int" } EQ_Contact(in1 := "PalletNGData".UnLoadingNGPallet.LockStatus, in2 := 4)
      I_Contact( "iNG_Button2" )
      Move(in := 1, out1 => "PalletNGData".UnLoadingNGPallet.LockStatus)
   END_RUNG
   // the same network as SCL:
   #_w1 := "AlwaysTRUE" AND "Station_Sys".Status.Run AND NOT "AutoProcessControl".Robot_3.NGPutFlag;
   #_w2 := #_w1 AND "AlwaysTRUE";
   #_w3 := #_w2 AND "Station_Sys".Manual.Mode AND "iNG_Button2";
   #_w4 := #_w3 AND ("PalletNGData".UnLoadingNGPallet.LockStatus = 1);
   #_w5 := #_w4 AND NOT "PalletNGData".P[4];   // rising edge
   "PalletNGData".P[4] := #_w4;
   IF #_w5 THEN
       "ST10Cylinder".Cy[12].Inout.ManualGoHome := TRUE;
       "ST10Cylinder".Cy[12].Inout.ManualGoWork := FALSE;
       "ST10_NGGate2_DB"."sSafetyGate UnlockRequest" := TRUE;
       "ST10_NGGate2_DB"."sSafetyGate LockRequest" := FALSE;
       "PalletNGData".UnLoadingNGPallet.LockStatus := 2;
   END_IF;
   #_w6 := #_w3 AND ("PalletNGData".UnLoadingNGPallet.LockStatus = 3) AND "PalletNGData".UnLoadingNGPallet.Interlock_1[2];
   #_w7 := #_w6 AND NOT "PalletNGData".P[5];   // rising edge
   "PalletNGData".P[5] := #_w6;
   IF #_w7 THEN
       "ST10Cylinder".Cy[12].Inout.ManualGoHome := FALSE;
       "ST10Cylinder".Cy[12].Inout.ManualGoWork := TRUE;
       "ST10_NGGate2_DB"."sSafetyGate UnlockRequest" := FALSE;
       "ST10_NGGate2_DB"."sSafetyGate LockRequest" := TRUE;
       "PalletNGData".UnLoadingNGPallet.LockStatus := 4;
   END_IF;
   #_w8 := #_w2 AND "Station_Sys".Auto.Mode;
   #_w9 := #_w8 AND "iNG_Button2";
   #_w10 := #_w9 AND ("PalletNGData".UnLoadingNGPallet.LockStatus = 1);
   #_w11 := #_w10 AND NOT "PalletNGData".P[6];   // rising edge
   "PalletNGData".P[6] := #_w10;
   IF #_w11 THEN "PalletNGData".UnLoadingNGPallet.OpenFlag := TRUE; END_IF;
   #_w12 := #_w9 AND ("PalletNGData".UnLoadingNGPallet.LockStatus = 3) AND "PalletNGData".UnLoadingNGPallet.Interlock_1[2];
   #_w13 := #_w12 AND NOT "PalletNGData".P[7];   // rising edge
   "PalletNGData".P[7] := #_w12;
   IF #_w13 THEN
       "ST10Cylinder".Cy[12].Inout.AutoGoHome := FALSE;
       "ST10Cylinder".Cy[12].Inout.AutoGoWork := TRUE;
       "ST10_NGGate2_DB"."sSafetyGate UnlockRequest" := FALSE;
       "ST10_NGGate2_DB"."sSafetyGate LockRequest" := TRUE;
       "PalletNGData".UnLoadingNGPallet.OpenFlag := FALSE;
       "PalletNGData".UnLoadingNGPallet.LockStatus := 4;
   END_IF;
   IF #_w8 AND "PalletNGData".UnLoadingNGPallet.OpenFlag AND "ST10_Flow15_FRobot_3_iDB".RobotTaskSelect.X AND "KukaRobot3_CtrlDB".sROBtoPLC.Sys.SO.ROB_STOPPED THEN
       "ST10Cylinder".Cy[12].Inout.AutoGoHome := TRUE;
       "ST10Cylinder".Cy[12].Inout.AutoGoWork := FALSE;
       "ST10_NGGate2_DB"."sSafetyGate UnlockRequest" := TRUE;
       "ST10_NGGate2_DB"."sSafetyGate LockRequest" := FALSE;
       "PalletNGData".UnLoadingNGPallet.LockStatus := 2;
   END_IF;
   IF #_w1 AND ("PalletNGData".UnLoadingNGPallet.LockStatus <> 1) AND ("PalletNGData".UnLoadingNGPallet.LockStatus <> 2) AND ("PalletNGData".UnLoadingNGPallet.LockStatus <> 3) AND ("PalletNGData".UnLoadingNGPallet.LockStatus <> 4) THEN
       "PalletNGData".UnLoadingNGPallet.LockStatus := 1;
   END_IF;
   IF #_w1 AND ("PalletNGData".UnLoadingNGPallet.LockStatus = 2) AND NOT "iNG_Button2" THEN
       "PalletNGData".UnLoadingNGPallet.LockStatus := 3;
   END_IF;
   IF #_w1 AND ("PalletNGData".UnLoadingNGPallet.LockStatus = 4) AND NOT "iNG_Button2" THEN
       "PalletNGData".UnLoadingNGPallet.LockStatus := 1;
   END_IF;
END_REGION

REGION Network 17: FlagReset
   RUNG wire#powerrail
      Contact( "AlwaysTRUE" )
      I_Contact( "Station_Sys".Auto.Mode )
      R_Coil( "PalletNGData".UnLoadingNGPallet.OpenFlag )
   END_RUNG
   // the same network as SCL:
   IF "AlwaysTRUE" AND NOT "Station_Sys".Auto.Mode THEN
       "PalletNGData".UnLoadingNGPallet.OpenFlag := FALSE;
   END_IF;
END_REGION

REGION Network 18: NG Door
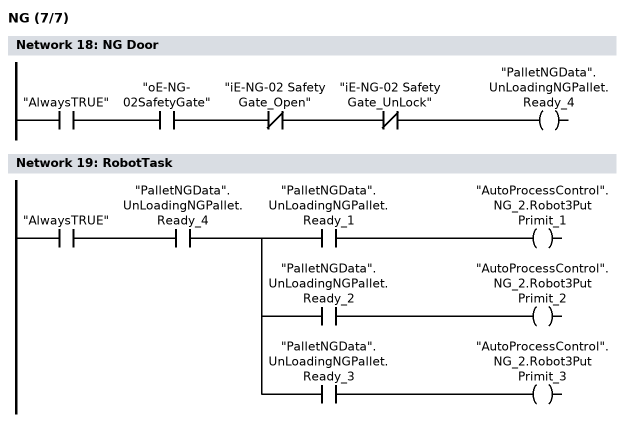
   RUNG wire#powerrail
      Contact( "AlwaysTRUE" )
      Contact( "oE-NG-02SafetyGate" )
      I_Contact( "iE-NG-02 Safety Gate_Open" )
      I_Contact( "iE-NG-02 Safety Gate_UnLock" )
      Coil( "PalletNGData".UnLoadingNGPallet.Ready_4 )
   END_RUNG
   // the same network as SCL:
   "PalletNGData".UnLoadingNGPallet.Ready_4 := "AlwaysTRUE" AND "oE-NG-02SafetyGate" AND NOT "iE-NG-02 Safety Gate_Open" AND NOT "iE-NG-02 Safety Gate_UnLock";
END_REGION

REGION Network 19: RobotTask
   RUNG wire#powerrail
      Contact( "AlwaysTRUE" )
      Contact( "PalletNGData".UnLoadingNGPallet.Ready_4 )
      wire#w1
      Contact( "PalletNGData".UnLoadingNGPallet.Ready_1 )
      Coil( "AutoProcessControl".NG_2.Robot3PutPrimit_1 )
   END_RUNG
   RUNG wire#w1
      Contact( "PalletNGData".UnLoadingNGPallet.Ready_2 )
      Coil( "AutoProcessControl".NG_2.Robot3PutPrimit_2 )
   END_RUNG
   RUNG wire#w1
      Contact( "PalletNGData".UnLoadingNGPallet.Ready_3 )
      Coil( "AutoProcessControl".NG_2.Robot3PutPrimit_3 )
   END_RUNG
   // the same network as SCL:
   #_w1 := "AlwaysTRUE" AND "PalletNGData".UnLoadingNGPallet.Ready_4;
   "AutoProcessControl".NG_2.Robot3PutPrimit_1 := #_w1 AND "PalletNGData".UnLoadingNGPallet.Ready_1;
   "AutoProcessControl".NG_2.Robot3PutPrimit_2 := #_w1 AND "PalletNGData".UnLoadingNGPallet.Ready_2;
   "AutoProcessControl".NG_2.Robot3PutPrimit_3 := #_w1 AND "PalletNGData".UnLoadingNGPallet.Ready_3;
END_REGION
END_FUNCTION_BLOCK
